// TIA Portal V19 export
TYPE "CTRL_DIFF"
   STRUCT
      status : Bool;
   END_STRUCT;
END_TYPE
